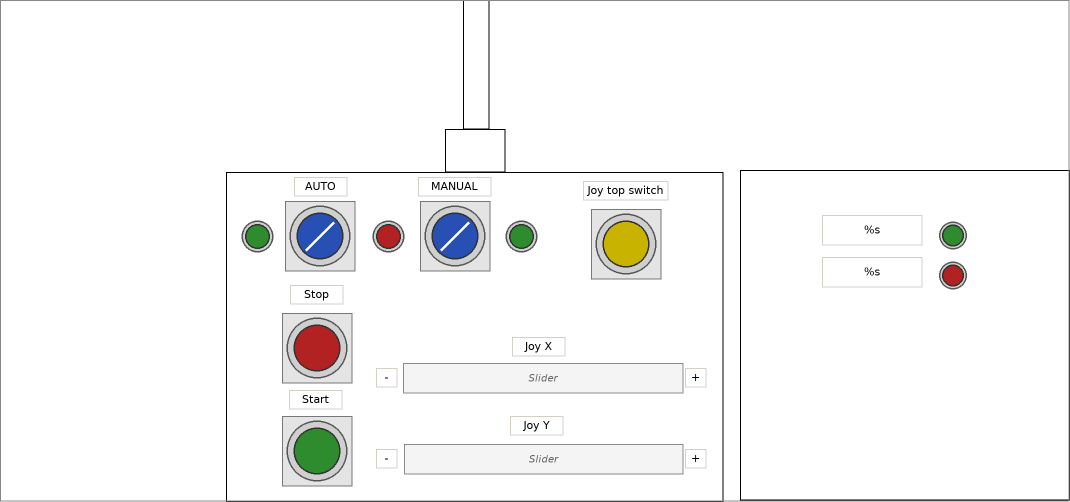
VISUALIZATION Visualization  // 1070x502
    RoundedRectangle (226,172 497x330)
    RotarySwitch (285,201 70x70), variable: G_Virtual_Input.bAuto, behaviour: TOGGLE, style: Switch-RotarySwitch-Blue
    PushSwitch (282,416 70x70), variable: G_Virtual_Input.bStart, behaviour: TOGGLE, style: Switch-PushSwitch-Green
    PushSwitch (282,313 70x70), variable: G_Virtual_Input.bStop, behaviour: TOGGLE, style: Switch-PushSwitch-Red
    RotarySwitch (420,201 70x70), variable: G_Virtual_Input.bManual, behaviour: TOGGLE, style: Switch-RotarySwitch-Blue
    Slider (404,444 279x30), variable: G_Virtual_Input.fJoyY, input disabled if: G_Virtual_Input.bJoyNotActive, scale 0..0
    Slider (403,363 280x30), variable: G_Virtual_Input.fJoyX, input disabled if: G_Virtual_Input.bJoyNotActive, scale 0..0
    Rectangle (445,129 60x43)
    Rectangle (463,0 26x129)
    Textfield (290,285 53x19), "Stop"
    Textfield (289,390 53x19), "Start"
    Textfield (512,337 53x19), "Joy X"
    Textfield (510,416 53x19), "Joy Y"
    PushSwitchLed (591,209 70x70), variable: G_Virtual_Input.bJoyActive, behaviour: TOGGLE, style: Switch-PushSwitchLed-Yellow
    Textfield (583,181 85x19), "Joy top switch"
    Textfield (685,368 21x19), "+"
    Textfield (685,449 21x19), "+"
    Textfield (376,449 21x19), "-"
    Textfield (376,368 21x19), "-"
    Textfield (294,177 53x19), "AUTO"
    Textfield (418,177 73x19), "MANUAL"
    RoundedRectangle (740,170 330x330)
    Label (756,214 63x30), "Mode:"
    Label (738,253 90x38), "Status:"
    Textfield (822,215 100x30), "%s", text variable: G_ControlBox.eMode
    Lamp1 (937,215 32x41), style: Lamp-Lamp1-Green
    Textfield (822,257 100x30), "%s", text variable: G_ControlBox.eStatus
    Lamp1 (937,255 32x41), variable: G_Virtual_Input.bStopping, style: Lamp-Lamp1-Red
    Lamp1 (239,216 37x41), variable: G_Virtual_Input.bAuto, style: Lamp-Lamp1-Green
    Lamp1 (370,216 37x41), variable: G_Virtual_Input.bOff, style: Lamp-Lamp1-Red
    Lamp1 (503,216 37x41), variable: G_Virtual_Input.bManual, style: Lamp-Lamp1-Green
END_VISUALIZATION

(* stored: Version 1.1.0.1, ProductVersion 3.1.4024.12
   Visu Visualization: Id {81918428-894a-4d31-8869-aaee674000f5} *)
